FUNCTION_BLOCK SmokeDetector
VAR_INPUT
	EN: BOOL;
	Input: REFERENCE TO AnalogInput;
	FireAlarm: REFERENCE TO AnalogAlarm;
	ServiceAlarm: REFERENCE TO AnalogAlarm;
END_VAR
VAR_OUTPUT
	ENO: BOOL;
END_VAR
VAR
END_VAR

END_FUNCTION_BLOCK

(* stored: Version 1.1.0.1, ProductVersion 3.1.4024.3
   POU SmokeDetector: Id {21482072-5996-45ed-abad-28da342bc882}, SpecialFunc None *)
